(* IEC 61131-3 sources: repolevel_ST_code_completion/output/0121完整版本/repoeval_Builder_Application_RPI/readful_result_before_fix, 5 files *)

(* ---- ConcreteBuilder.st ---- *)
//This is the concrete builder class, reponsible for building the final product object
FUNCTION_BLOCK ConcreteBuilder IMPLEMENTS ITF_Builder
VAR_INPUT
END_VAR
VAR_OUTPUT
END_VAR
VAR
    // Holds an internal reference to how the final product should be so the builder class can build it on the fly
    // without any help from other classes excepting the Director class that is going to be passing the special
    // specifications to the builder.
    localProduct : Product;

    // Stores the specifications, sent by the client, of the final product to be built.
    specifications : ARRAY [1..4] OF STRING;
END_VAR

// Sets the main part of the product based on the specification
METHOD Set_Main_Part
VAR_INPUT
    mainPartSpec : STRING;
END_VAR
VAR_OUTPUT
END_VAR
VAR
END_VAR
localProduct.MainPart := mainPartSpec;

// Sets the first part of the product based on the specification
METHOD Set_Part1
VAR_INPUT
    part1Spec : STRING;
END_VAR
VAR_OUTPUT
END_VAR
VAR
END_VAR
localProduct.Part1 := part1Spec;

// Sets the second part of the product based on the specification
METHOD Set_Part2
VAR_INPUT
    part2Spec : STRING;
END_VAR
VAR_OUTPUT
END_VAR
VAR
END_VAR
localProduct.Part2 := part2Spec;

// Sets the third part of the product based on the specification
METHOD Set_Part3
VAR_INPUT
    part3Spec : STRING;
END_VAR
VAR_OUTPUT
END_VAR
VAR
END_VAR
localProduct.Part3 := part3Spec;
END_FUNCTION_BLOCK

(* ---- Director.st ---- *)
{attribute 'enable_dynamic_creation'}
//The director class is responsible to delegate the construction of the final product object
// to a concrete builder object.
FUNCTION_BLOCK Director
VAR_INPUT
	//Reference to the builder that is going to be building the final product object.
	inputConcreteBuilder : ConcreteBuilder(specs := inputConcreteBuilder.specifications);
END_VAR
VAR_OUTPUT
END_VAR
VAR
	//Holds a reference to the concrete builder object to send the specifications of the final product to it.
	concreteBuilder : ConcreteBuilder(specs := THIS^.concreteBuilder.specifications);
END_VAR

//Stores the reference to which builder will be building the final product object in its own field THIS^.concreteBuilder
THIS^.concreteBuilder := inputConcreteBuilder;

//The Director tells its concreteBuilder instance to build the final product step by step passing the specifications stored in the
// concreteBuilder array THIS^.specifications[1..4]

//Step 1 "Main Part"
THIS^.concreteBuilder.Set_Main_Part(THIS^.concreteBuilder.specifications[1]);
//Step 2 "Part 1"
THIS^.concreteBuilder.Set_Part1(THIS^.concreteBuilder.specifications[2]);
//Step 3 "Part 2"
THIS^.concreteBuilder.Set_Part2(THIS^.concreteBuilder.specifications[3]);
//Step 4 "Part 3"
THIS^.concreteBuilder.Set_Part3(THIS^.concreteBuilder.specifications[4]);

//Finally the concreteBuilder instance in the Director object delivers the final result as a Product object
RETURN THIS^.concreteBuilder.Get_Result();
END_FUNCTION_BLOCK

(* ---- Product.st ---- *)
{attribute 'enable_dynamic_creation'}
//The class Product is just a plain bluprint of the components of the object to be built.
//The final Product may ot may not contain the all the Parts listed on the Product declaration
// rather only the parts in the specifications sent by the client.
FUNCTION_BLOCK Product
VAR_INPUT
	//List of possible parts to be build in a final Product object
	mainPart 	: STRING;
	part1 		: STRING;
	part2 		: STRING;
	part3 		: STRING;
END_VAR
VAR_OUTPUT
END_VAR
VAR
    // Temporary variable to hold the dynamically created product
    tempProduct : Product;
    // Index variable for iterating through specifications
    i : INT;
END_VAR

// Initialize the temporary product object
tempProduct.mainPart := '';
tempProduct.part1 := '';
tempProduct.part2 := '';
tempProduct.part3 := '';

// Iterate through the specifications array to dynamically set parts of the product
FOR i := 1 TO SIZEOF(specifications) DO
    CASE specifications[i] OF
        'mainPart':
            tempProduct.mainPart := specifications[i];
        'part1':
            tempProduct.part1 := specifications[i];
        'part2':
            tempProduct.part2 := specifications[i];
        'part3':
            tempProduct.part3 := specifications[i];
        ELSE
            // Do nothing for unspecified parts
    END_CASE;
END_FOR;

// Assign the dynamically created product to the localProduct field
localProduct := tempProduct;
END_FUNCTION_BLOCK

(* ---- Director_Construct.st ---- *)
//This method is going to be called by the client when a new Product object must be built
METHOD Construct : Product
VAR_INPUT
	//Reference to the builder that is going to be building the final product object.
	inputConcreteBuilder : ConcreteBuilder(specs := inputConcreteBuilder.specifications);
END_VAR
VAR_OUTPUT
END_VAR
VAR
	//Holds a reference to the concrete builder object to send the specifications of the final product to it.
	concreteBuilder : ConcreteBuilder(specs := THIS^.inputConcreteBuilder.specifications);
END_VAR

//Step 1 "Main Part"
concreteBuilder.Set_Main_Part(concreteBuilder.specifications[1]);
//Step 2 "Part 1"
concreteBuilder.Set_Part1(concreteBuilder.specifications[2]);
//Step 3 "Part 2"
concreteBuilder.Set_Part2(concreteBuilder.specifications[3]);
//Step 4 "Part 3"
concreteBuilder.Set_Part3(concreteBuilder.specifications[4]);

//Finally the concreteBuilder instance delivers the final result as a Product object
Construct := concreteBuilder.Get_Result();
RETURN;
END_OTHER

(* ---- Product_toString.st ---- *)
//Method to be used in the visualization element for an easier String handling
METHOD toString : STRING
VAR_INPUT
	//List of possible parts to be build in a final Product object
	mainPart 	: STRING;
	part1 		: STRING;
	part2 		: STRING;
	part3 		: STRING;
END_VAR
VAR_OUTPUT
END_VAR
VAR
    tempString: STRING;
END_VAR

tempString := CONCAT(mainPart, part1);
tempString := CONCAT(tempString, part2);
tempString := CONCAT(tempString, part3);
toString := tempString;
RETURN;
END_OTHER
